TYPE T_Generic : __SYSTEM.AnyType; END_TYPE

(* stored: Version 1.1.0.1, ProductVersion 3.1.4024.4
   DUT T_Generic: Id {7033d824-d54f-0bc1-03c8-53f60c07df9c} *)
